Staubli VAL3: Prefix.dtx

mdesc mNomSpeed
public num nLength
public num nData[4]
